# EPICS autosave request: iocBoot/ioc13SmarAct1/auto_settings.req
file "CARS_motor_settings.req",         P=$(P), M=m1
file "CARS_motor_settings.req",         P=$(P), M=m2
